FUNCTION_BLOCK JackDecode_New (* Basic Function Block Type *)
  (* Standard: 61499-2 *)
  (* Version 0.0, 11/3/2020, prana, nxtControl GmbH, Template *)
  PACKAGE Main;
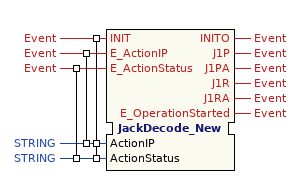
  EVENT_INPUT
    INIT WITH ActionIP, ActionStatus; (* Initialization Request *)
    E_ActionIP WITH ActionIP; (* Normal Execution Request *)
    E_ActionStatus WITH ActionStatus;
  END_EVENT
  EVENT_OUTPUT
    INITO; (* Initialization Confirm *)
    J1P; (* Execution Confirmation *)
    J1PA;
    J1R;
    J1RA;
    E_OperationStarted;
  END_EVENT
  VAR_INPUT
    ActionIP : STRING; (* Input event qualifier *)
    ActionStatus : STRING;
  END_VAR
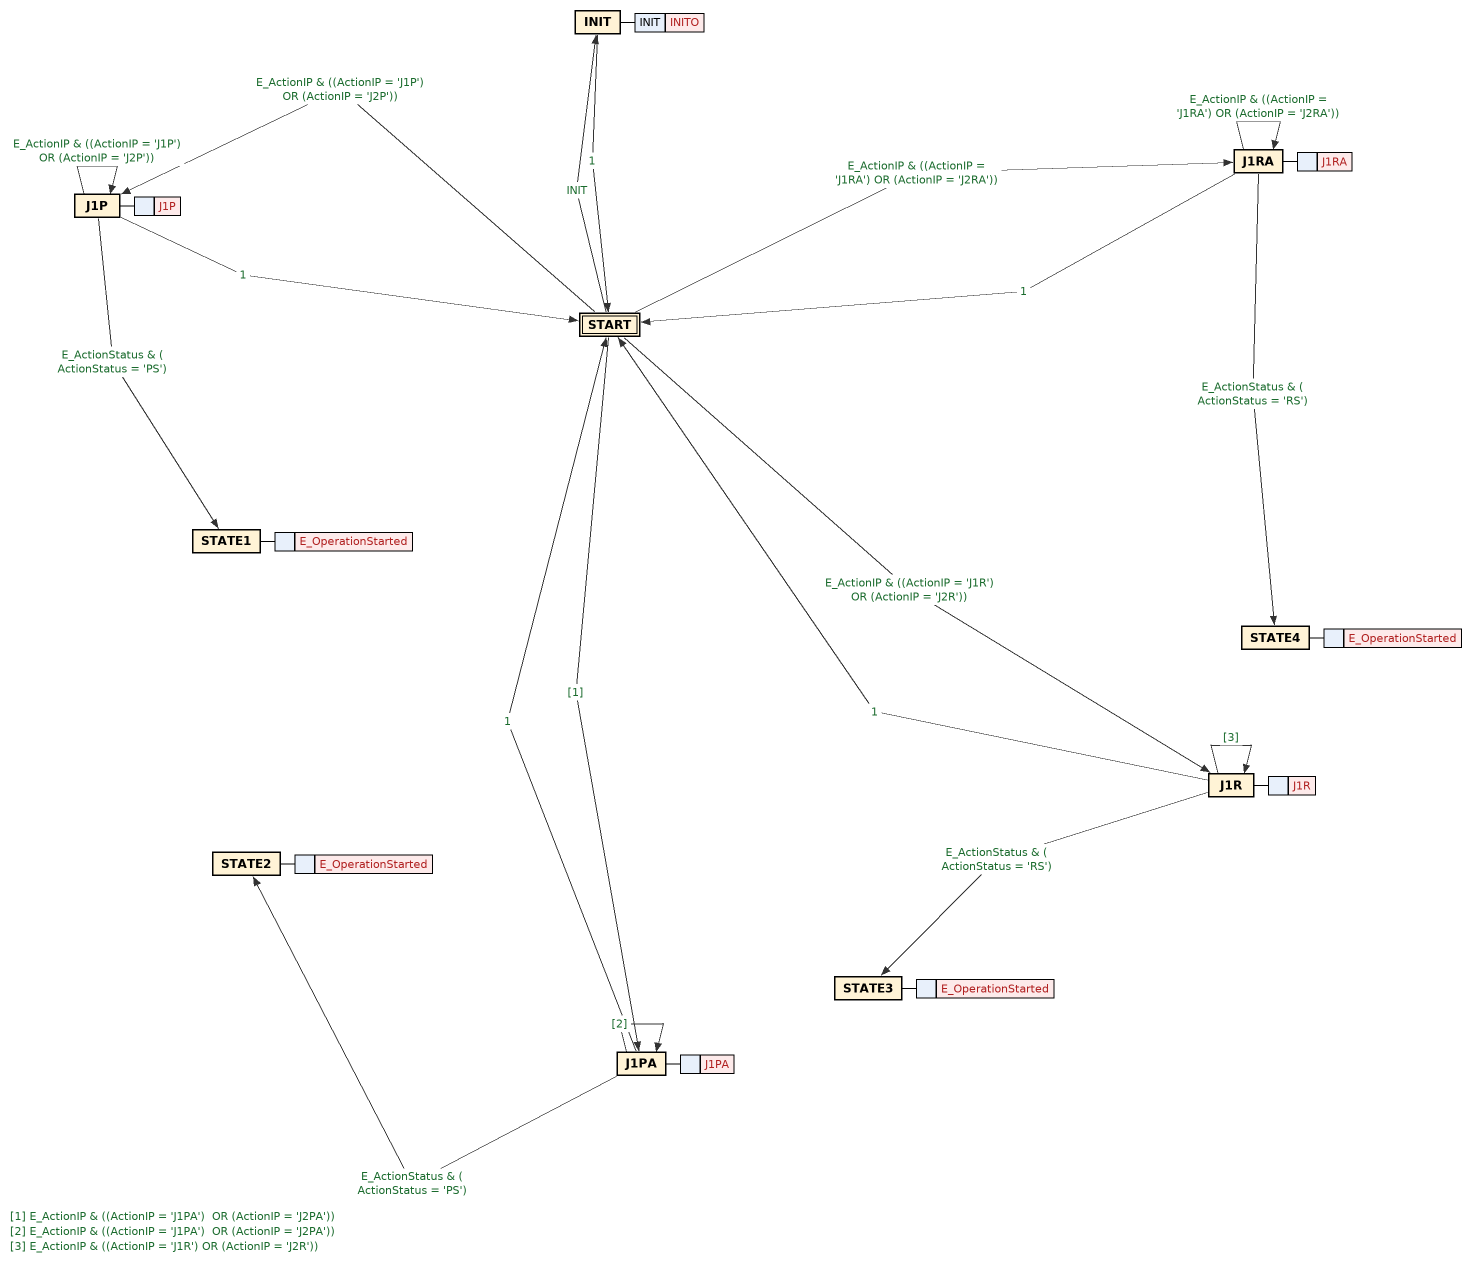
  EC_STATES
    START; (* Initial State *)
    INIT : INIT -> INITO; (* Initialization *)
    J1P : -> J1P;
    J1PA : -> J1PA;
    J1R : -> J1R;
    J1RA : -> J1RA;
    STATE1 : -> E_OperationStarted;
    STATE2 : -> E_OperationStarted;
    STATE3 : -> E_OperationStarted;
    STATE4 : -> E_OperationStarted;
  END_STATES
  EC_TRANSITIONS
    START TO INIT := INIT;
    INIT TO START := 1;
    START TO J1P := E_ActionIP & ((ActionIP = 'J1P') OR (ActionIP = 'J2P'));
    START TO J1PA := E_ActionIP & ((ActionIP = 'J1PA')  OR (ActionIP = 'J2PA'));
    START TO J1R := E_ActionIP & ((ActionIP = 'J1R') OR (ActionIP = 'J2R'));
    START TO J1RA := E_ActionIP & ((ActionIP = 'J1RA') OR (ActionIP = 'J2RA'));
    J1P TO START := 1;
    J1PA TO START := 1;
    J1R TO START := 1;
    J1RA TO START := 1;
    J1P TO STATE1 := E_ActionStatus & ( ActionStatus = 'PS');
    J1PA TO STATE2 := E_ActionStatus & ( ActionStatus = 'PS');
    J1R TO STATE3 := E_ActionStatus & ( ActionStatus = 'RS');
    J1RA TO STATE4 := E_ActionStatus & ( ActionStatus = 'RS');
    J1P TO J1P := E_ActionIP & ((ActionIP = 'J1P') OR (ActionIP = 'J2P'));
    J1PA TO J1PA := E_ActionIP & ((ActionIP = 'J1PA')  OR (ActionIP = 'J2PA'));
    J1R TO J1R := E_ActionIP & ((ActionIP = 'J1R') OR (ActionIP = 'J2R'));
    J1RA TO J1RA := E_ActionIP & ((ActionIP = 'J1RA') OR (ActionIP = 'J2RA'));
  END_TRANSITIONS
  ALGORITHM INIT IN ST: (* Initialization algorithm *)
;
  END_ALGORITHM
  ALGORITHM REQ IN ST: (* Normally executed algorithm *)
;
  END_ALGORITHM
END_FUNCTION_BLOCK
